// TIA Portal V18 export
// export: Created 2026-06-09T02:36:18.0488678Z, ExportSetting WithDefaults, DisplayName Totally Integrated Automation Portal, DisplayVersion V18, DisplayName TIA Portal Openness, DisplayVersion V18, DisplayName TIA Portal Version Control Interface, DisplayVersion V18, DisplayName STEP 7 Professional, DisplayVersion V18, DisplayName STEP 7 Safety, DisplayVersion V18, DisplayName WinCC Professional, DisplayVersion V18
ORGANIZATION_BLOCK "Main"   // OB1, LAD, ProgramCycle
TITLE = "Main Program Sweep (Cycle)"
{ S7_Optimized_Access := 'TRUE' }
VERSION : 0.1
// stored: AutoNumber true, IsIECCheckEnabled false, SetENOAutomatically false
   VAR_INPUT
      Initial_Call : Bool;   // Initial call of this OB
      Remanence : Bool;   // =True, if remanent data are available
   END_VAR
   VAR_TEMP   // added for the SCL form of the ladder/FBD networks
      _w1 : Bool;
   END_VAR
BEGIN

REGION Network 1
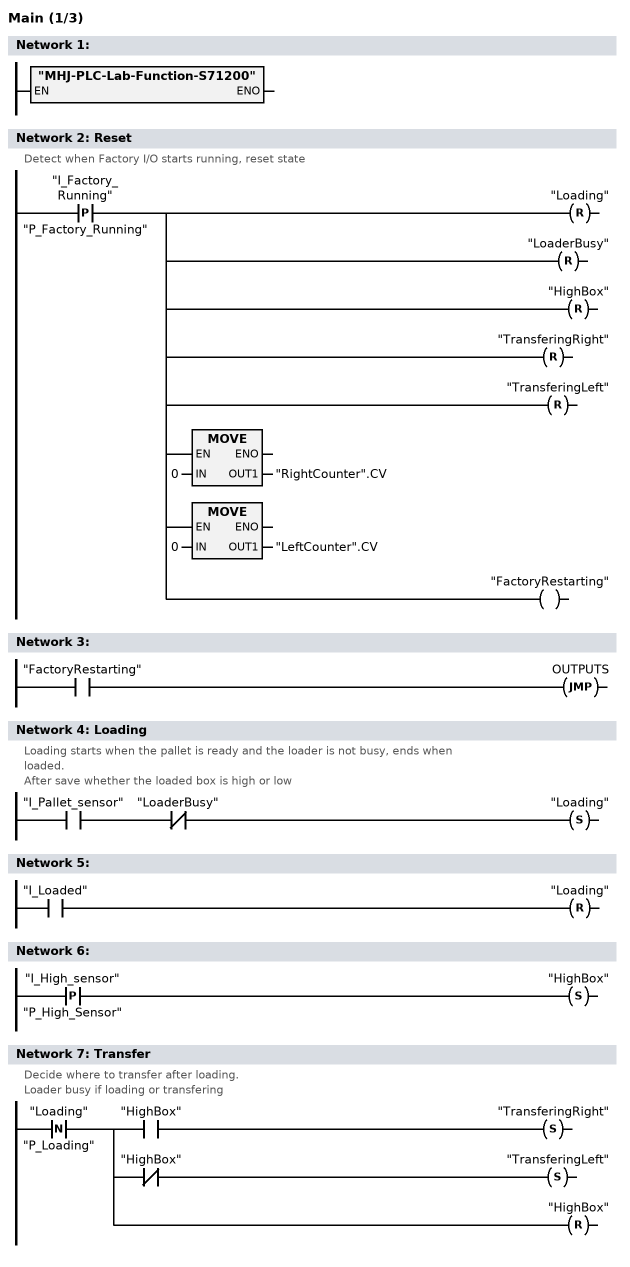
   RUNG wire#powerrail
      "MHJ-PLC-Lab-Function-S71200"()
   END_RUNG
   // the same network as SCL:
   "MHJ-PLC-Lab-Function-S71200"();
END_REGION

REGION Network 2: Reset
   // Detect when Factory I/O starts running, reset state
   RUNG wire#powerrail
      P_Contact(operand := "I_Factory_Running", bit := "P_Factory_Running")
      wire#w1
      R_Coil( "Loading" )
   END_RUNG
   RUNG wire#w1
      R_Coil( "LoaderBusy" )
   END_RUNG
   RUNG wire#w1
      R_Coil( "HighBox" )
   END_RUNG
   RUNG wire#w1
      R_Coil( "TransferingRight" )
   END_RUNG
   RUNG wire#w1
      R_Coil( "TransferingLeft" )
   END_RUNG
   RUNG wire#w1
      { S7_GenerateENO := "TRUE" } Move(in := 0, out1 => "RightCounter".CV)
   END_RUNG
   RUNG wire#w1
      { S7_GenerateENO := "TRUE" } Move(in := 0, out1 => "LeftCounter".CV)
   END_RUNG
   RUNG wire#w1
      Coil( "FactoryRestarting" )
   END_RUNG
   // the same network as SCL:
   #_w1 := "I_Factory_Running" AND NOT "P_Factory_Running";   // rising edge of "I_Factory_Running"
   "P_Factory_Running" := "I_Factory_Running";
   IF #_w1 THEN
       "Loading" := FALSE;
       "LoaderBusy" := FALSE;
       "HighBox" := FALSE;
       "TransferingRight" := FALSE;
       "TransferingLeft" := FALSE;
       "RightCounter".CV := 0;
       "LeftCounter".CV := 0;
   END_IF;
   "FactoryRestarting" := #_w1;
END_REGION

REGION Network 3
   RUNG wire#powerrail
      Contact( "FactoryRestarting" )
      JumpCoil( OUTPUTS )
   END_RUNG
   // the same network as SCL:
   IF "FactoryRestarting" THEN GOTO OUTPUTS; END_IF;
END_REGION

REGION Network 4: Loading
   // Loading starts when the pallet is ready and the loader is not busy, ends when 
   // loaded.
   // After save whether the loaded box is high or low
   RUNG wire#powerrail
      Contact( "I_Pallet_sensor" )
      I_Contact( "LoaderBusy" )
      S_Coil( "Loading" )
   END_RUNG
   // the same network as SCL:
   IF "I_Pallet_sensor" AND NOT "LoaderBusy" THEN "Loading" := TRUE; END_IF;
END_REGION

REGION Network 5
   RUNG wire#powerrail
      Contact( "I_Loaded" )
      R_Coil( "Loading" )
   END_RUNG
   // the same network as SCL:
   IF "I_Loaded" THEN "Loading" := FALSE; END_IF;
END_REGION

REGION Network 6
   RUNG wire#powerrail
      P_Contact(operand := "I_High_sensor", bit := "P_High_Sensor")
      S_Coil( "HighBox" )
   END_RUNG
   // the same network as SCL:
   #_w1 := "I_High_sensor" AND NOT "P_High_Sensor";   // rising edge of "I_High_sensor"
   "P_High_Sensor" := "I_High_sensor";
   IF #_w1 THEN "HighBox" := TRUE; END_IF;
END_REGION

REGION Network 7: Transfer
   // Decide where to transfer after loading.
   // Loader busy if loading or transfering
   RUNG wire#powerrail
      N_Contact(operand := "Loading", bit := "P_Loading")
      wire#w1
      Contact( "HighBox" )
      S_Coil( "TransferingRight" )
   END_RUNG
   RUNG wire#w1
      I_Contact( "HighBox" )
      S_Coil( "TransferingLeft" )
   END_RUNG
   RUNG wire#w1
      R_Coil( "HighBox" )
   END_RUNG
   // the same network as SCL:
   #_w1 := NOT "Loading" AND "P_Loading";   // falling edge of "Loading"
   "P_Loading" := "Loading";
   IF #_w1 AND "HighBox" THEN "TransferingRight" := TRUE; END_IF;
   IF #_w1 AND NOT "HighBox" THEN "TransferingLeft" := TRUE; END_IF;
   IF #_w1 THEN "HighBox" := FALSE; END_IF;
END_REGION

REGION Network 8
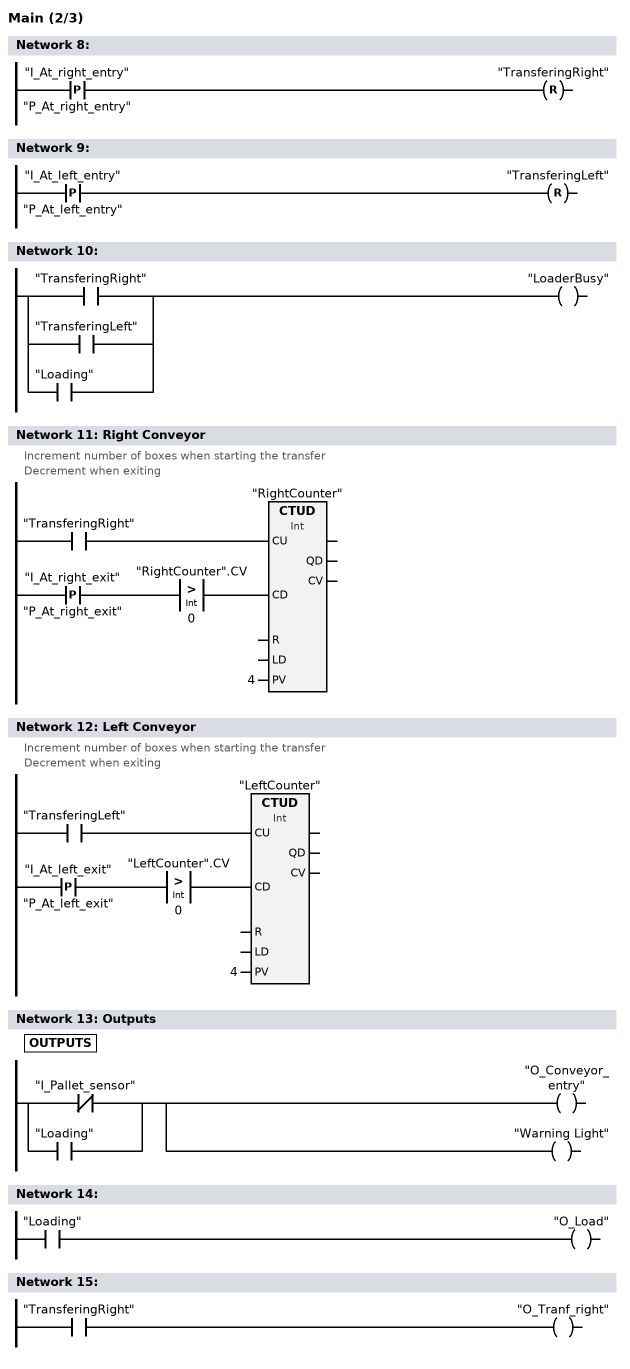
   RUNG wire#powerrail
      P_Contact(operand := "I_At_right_entry", bit := "P_At_right_entry")
      R_Coil( "TransferingRight" )
   END_RUNG
   // the same network as SCL:
   #_w1 := "I_At_right_entry" AND NOT "P_At_right_entry";   // rising edge of "I_At_right_entry"
   "P_At_right_entry" := "I_At_right_entry";
   IF #_w1 THEN "TransferingRight" := FALSE; END_IF;
END_REGION

REGION Network 9
   RUNG wire#powerrail
      P_Contact(operand := "I_At_left_entry", bit := "P_At_left_entry")
      R_Coil( "TransferingLeft" )
   END_RUNG
   // the same network as SCL:
   #_w1 := "I_At_left_entry" AND NOT "P_At_left_entry";   // rising edge of "I_At_left_entry"
   "P_At_left_entry" := "I_At_left_entry";
   IF #_w1 THEN "TransferingLeft" := FALSE; END_IF;
END_REGION

REGION Network 10
   RUNG wire#powerrail
      Contact( "TransferingRight" )
      wire#w1
      Coil( "LoaderBusy" )
   END_RUNG
   RUNG wire#powerrail
      Contact( "TransferingLeft" )
   END_RUNG wire#w1
   RUNG wire#powerrail
      Contact( "Loading" )
   END_RUNG wire#w1
   // the same network as SCL:
   "LoaderBusy" := "TransferingRight" OR "TransferingLeft" OR "Loading";
END_REGION

REGION Network 11: Right Conveyor
   // Increment number of boxes when starting the transfer
   // Decrement when exiting
   RUNG wire#powerrail
      Contact( "TransferingRight" )
      { S7_Templates := "value_type := Int" } "RightCounter".CTUD(cd := wire#w1, r :=, ld :=, pv := 4, qd =>, cv =>)
   END_RUNG
   RUNG wire#powerrail
      P_Contact(operand := "I_At_right_exit", bit := "P_At_right_exit")
      { S7_Templates := "SrcType := Int" } GT_Contact(in1 := "RightCounter".CV, in2 := 0)
   END_RUNG wire#w1
   // the same network as SCL:
   #_w1 := "I_At_right_exit" AND NOT "P_At_right_exit";   // rising edge of "I_At_right_exit"
   "P_At_right_exit" := "I_At_right_exit";
   "RightCounter".CTUD(CU := "TransferingRight", CD := #_w1 AND ("RightCounter".CV > 0), PV := 4);
END_REGION

REGION Network 12: Left Conveyor
   // Increment number of boxes when starting the transfer
   // Decrement when exiting
   RUNG wire#powerrail
      Contact( "TransferingLeft" )
      { S7_Templates := "value_type := Int" } "LeftCounter".CTUD(cd := wire#w1, r :=, ld :=, pv := 4, qd =>, cv =>)
   END_RUNG
   RUNG wire#powerrail
      P_Contact(operand := "I_At_left_exit", bit := "P_At_left_exit")
      { S7_Templates := "SrcType := Int" } GT_Contact(in1 := "LeftCounter".CV, in2 := 0)
   END_RUNG wire#w1
   // the same network as SCL:
   #_w1 := "I_At_left_exit" AND NOT "P_At_left_exit";   // rising edge of "I_At_left_exit"
   "P_At_left_exit" := "I_At_left_exit";
   "LeftCounter".CTUD(CU := "TransferingLeft", CD := #_w1 AND ("LeftCounter".CV > 0), PV := 4);
END_REGION

REGION Network 13: Outputs
   Label( OUTPUTS )
   RUNG wire#powerrail
      I_Contact( "I_Pallet_sensor" )
      wire#w1
      Coil( "O_Conveyor_entry" )
   END_RUNG
   RUNG wire#powerrail
      Contact( "Loading" )
   END_RUNG wire#w1
   RUNG wire#w1
      Coil( "Warning Light" )
   END_RUNG
   // the same network as SCL:
   OUTPUTS:
   "O_Conveyor_entry" := NOT "I_Pallet_sensor" OR "Loading";
   "Warning Light" := "O_Conveyor_entry";
END_REGION

REGION Network 14
   RUNG wire#powerrail
      Contact( "Loading" )
      Coil( "O_Load" )
   END_RUNG
   // the same network as SCL:
   "O_Load" := "Loading";
END_REGION

REGION Network 15
   RUNG wire#powerrail
      Contact( "TransferingRight" )
      Coil( "O_Tranf_right" )
   END_RUNG
   // the same network as SCL:
   "O_Tranf_right" := "TransferingRight";
END_REGION

REGION Network 16
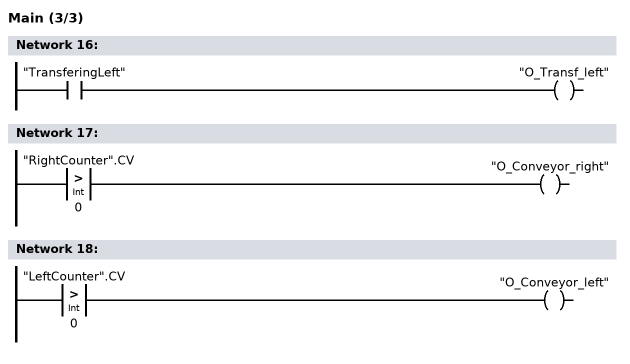
   RUNG wire#powerrail
      Contact( "TransferingLeft" )
      Coil( "O_Transf_left" )
   END_RUNG
   // the same network as SCL:
   "O_Transf_left" := "TransferingLeft";
END_REGION

REGION Network 17
   RUNG wire#powerrail
      { S7_Templates := "SrcType := Int" } GT_Contact(in1 := "RightCounter".CV, in2 := 0)
      Coil( "O_Conveyor_right" )
   END_RUNG
   // the same network as SCL:
   "O_Conveyor_right" := "RightCounter".CV > 0;
END_REGION

REGION Network 18
   RUNG wire#powerrail
      { S7_Templates := "SrcType := Int" } GT_Contact(in1 := "LeftCounter".CV, in2 := 0)
      Coil( "O_Conveyor_left" )
   END_RUNG
   // the same network as SCL:
   "O_Conveyor_left" := "LeftCounter".CV > 0;
END_REGION
END_ORGANIZATION_BLOCK
